// TwinCAT 3 PLC project AdsStaticNetIdEx
// ProgramVersion: 3.1.4023.0
// libraries:
//   Tc2_DataExchange, * (Beckhoff Automation GmbH)
//   Tc2_Standard, * (Beckhoff Automation GmbH)
//   Tc2_System, * (Beckhoff Automation GmbH)
//   Tc2_Utilities, * (Beckhoff Automation GmbH)
//   Tc3_BA_Common, * (Beckhoff Automation GmbH)
//   Tc3_Module, * (Beckhoff Automation GmbH)
// project tree:
//   DUTs/ AdsData.TcDUT (not stored), AdsMessageQueue.TcPOU (not stored), AdsMessage.TcDUT (not stored), AdsSocket.TcPOU, AreaNum.TcDUT (not stored), EventsEnum.TcTLEO (not stored)
//   GVLs/ LocalSocket.TcGVL, Sockets.TcGVL
//   / PlcTask.TcTTO (not stored)
//   POUs/ AdsTcpUnitEx.TcPOU (not stored), BufferIsEmpty.TcPOU (not stored), BytesToString.TcPOU (not stored), MAIN.TcPOU (not stored)

// ---- GVLs/LocalSocket.TcGVL
//{attribute 'qualified_only'}
VAR_GLOBAL CONSTANT
	PrgName : STRING := TO_STRING(AreaNum.AREA_4);
	AmsNetId : T_AmsNetId := '2.0.131.216.1.1';
	AmsPort : T_AmsPort := 851;
END_VAR

// ---- GVLs/Sockets.TcGVL
//{attribute 'qualified_only'}
VAR_GLOBAL
	AREA_1 : AdsSocket := (PrgName := 'AREA_1', AmsNetId := '1.0.131.216.1.1', AmsPort := 851);
	AREA_2 : AdsSocket := (PrgName := 'AREA_2', AmsNetId := '2.0.131.216.1.1', AmsPort := 851);
	AREA_3 : AdsSocket := (PrgName := 'AREA_3', AmsNetId := '3.0.131.216.1.1', AmsPort := 851);
	AREA_4 : AdsSocket := (PrgName := 'AREA_4', AmsNetId := ''(*'4.0.131.216.1.1'*), AmsPort := 851);
	AREA_5 : AdsSocket := (PrgName := 'AREA_5', AmsNetId := '5.0.131.216.1.1', AmsPort := 851);
	AREA_6 : AdsSocket := (PrgName := 'AREA_6', AmsNetId := '6.0.131.216.1.1', AmsPort := 851);
	adsMajorNetwork : AdsTcpUnitEx;
END_VAR
VAR_GLOBAL
	SUBAREA_4_1 : AdsSocket := (PrgName := 'SUBAREA_4_1', AmsNetId := '4.1.113.174.1.1', AmsPort := 851);
	SUBAREA_4_2 : AdsSocket := (PrgName := 'SUBAREA_4_2', AmsNetId := '4.2.113.174.1.1', AmsPort := 851);
	SUBAREA_4_3 : AdsSocket := (PrgName := 'SUBAREA_4_3', AmsNetId := '4.3.113.174.1.1', AmsPort := 851);
	SUBAREA_4_4 : AdsSocket := (PrgName := 'SUBAREA_4_4', AmsNetId := '4.4.113.174.1.1', AmsPort := 851);
	SUBAREA_4_5 : AdsSocket := (PrgName := 'SUBAREA_4_5', AmsNetId := '4.5.113.174.1.1', AmsPort := 851);
	SUBAREA_4_6 : AdsSocket := (PrgName := 'SUBAREA_4_6', AmsNetId := '4.6.113.174.1.1', AmsPort := 851);
	SUBAREA_4_7 : AdsSocket := (PrgName := 'SUBAREA_4_7', AmsNetId := '4.7.113.174.1.1', AmsPort := 851);
	SUBAREA_4_8 : AdsSocket := (PrgName := 'SUBAREA_4_8', AmsNetId := '4.8.113.174.1.1', AmsPort := 851);
	SUBAREA_4_9 : AdsSocket := (PrgName := 'SUBAREA_4_9', AmsNetId := '4.9.113.174.1.1', AmsPort := 851);
	adsLocalNetwork : AdsTcpUnitEx;
END_VAR
VAR_GLOBAL CONSTANT
	numSockets : INT := 6;
	numSubarea4Sockets : INT := 9;
END_VAR

// ---- DUTs/AdsSocket.TcPOU
FUNCTION_BLOCK AdsSocket
VAR_INPUT
END_VAR
VAR_OUTPUT
	//descriptive string for the name of the running program, may or may not be used
	PrgName : STRING;
	
	(*
	AmsNetId should be in the following format for ALL Beckhoff PLCs in the network:
		<area number> . <subarea number (0 for master PLC)> .131.216.1.1
		panel PCs to be assigned 113.174 instead of 131.216
			2.0.131.216.1.1 - Area 2, master controller
			4.3.113.174.1.1 - Area 4, manual station 3 panel PC
	*)
	AmsNetId : T_AmsNetId;
	
	//for now, use ADS port 851 for communication
	AmsPort : T_AmsPort;
END_VAR
VAR_OUTPUT
	receivingData : AdsData;
	sendingData : AdsData;
	
	readBusy : BOOL;
	readError : BOOL;
	readErrorId : UDINT;
	
	writeBusy : BOOL;
	writeError : BOOL;
	writeErrorId : UDINT;
END_VAR
VAR	
	adsWriteSymbol : FB_WriteAdsSymByName;
	adsReadSymbol : FB_ReadAdsSymByName;
END_VAR
VAR
	targetSocket : STRING;
	clearing : BOOL;
END_VAR
(*
TCP-style ADS connection that only writes to a buffer in the recipient's AdsTcpUnit module
*)

//write into the recipient's allocated socket for this system
targetSocket := CONCAT('Sockets.', LocalSocket.PrgName);

//only toggles if data has contents, otherwise remains false
adsWriteSymbol.bWrite := NOT BufferIsEmpty(sendingData.binaryData) AND NOT adsWriteSymbol.bWrite;

blocks();

IF NOT adsWriteSymbol.bBusy THEN
	MEMSET(ADR(sendingData), 0, SIZEOF(sendingData));
END_IF

METHOD PRIVATE blocks : BOOL
VAR_INPUT
END_VAR
adsReadSymbol(
	bRead:= , 
	sNetId:= AmsNetId, 
	nPort:= AmsPort, 
	sVarName:= , 
	nDestAddr:= , 
	nLen:= , 
	tTimeout:= , 
	eComMode:= , 
	bClearOnError:= , 
	bBusy=> readBusy, 
	bError=> readError, 
	nErrorId=> readErrorId);
	
adsWriteSymbol(
	bWrite:= , 
	sNetId:= AmsNetId, 
	nPort:= AmsPort, 
	sVarName:= CONCAT(targetSocket, '.receivingData'), 
	nSrcAddr:= ADR(sendingData), 
	nLen:= SIZEOF(sendingData), 
	tTimeout:= , 
	eComMode:= eAdsComModeSecureCom, 
	bBusy=> writeBusy, 
	bError=> writeError, 
	nErrorId=> writeErrorId);
END_METHOD

METHOD send : BOOL
VAR_INPUT
	data : REFERENCE TO AdsData;
END_VAR
sendingData := data;
END_METHOD

END_FUNCTION_BLOCK
